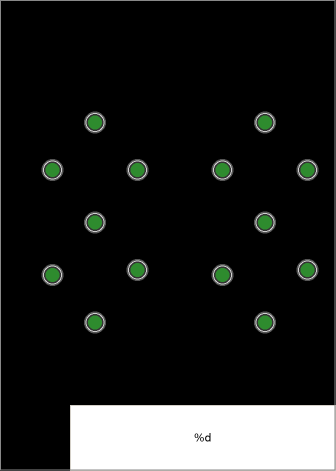
VISUALIZATION sevenSegmentDisplay  // 336x471
    Lamp1 (60,110 70x25), variable: sevenSegProg.digit1Decoder.decodedDigit[0], style: Lamp-Lamp1-Green
    Lamp1 (125,135 25x70), variable: sevenSegProg.digit1Decoder.decodedDigit[1], style: Lamp-Lamp1-Green
    Lamp1 (40,135 25x70), variable: sevenSegProg.digit1Decoder.decodedDigit[5], style: Lamp-Lamp1-Green
    Lamp1 (60,210 70x25), variable: sevenSegProg.digit1Decoder.decodedDigit[6], style: Lamp-Lamp1-Green
    Lamp1 (60,310 70x25), variable: sevenSegProg.digit1Decoder.decodedDigit[3], style: Lamp-Lamp1-Green
    Lamp1 (125,235 25x70), variable: sevenSegProg.digit1Decoder.decodedDigit[2], style: Lamp-Lamp1-Green
    Lamp1 (40,240 25x70), variable: sevenSegProg.digit1Decoder.decodedDigit[4], style: Lamp-Lamp1-Green
    Textfield (70,405 266x66), "%d", text variable: sevenSegProg.inputDigit
        OnMouseClick: write sevenSegProg.inputDigit via Default
    Lamp1 (230,110 70x25), variable: sevenSegProg.digit2Decoder.decodedDigit[0], style: Lamp-Lamp1-Green
    Lamp1 (295,135 25x70), variable: sevenSegProg.digit2Decoder.decodedDigit[1], style: Lamp-Lamp1-Green
    Lamp1 (210,135 25x70), variable: sevenSegProg.digit2Decoder.decodedDigit[5], style: Lamp-Lamp1-Green
    Lamp1 (230,210 70x25), variable: sevenSegProg.digit2Decoder.decodedDigit[6], style: Lamp-Lamp1-Green
    Lamp1 (230,310 70x25), variable: sevenSegProg.digit2Decoder.decodedDigit[3], style: Lamp-Lamp1-Green
    Lamp1 (295,235 25x70), variable: sevenSegProg.digit2Decoder.decodedDigit[2], style: Lamp-Lamp1-Green
    Lamp1 (210,240 25x70), variable: sevenSegProg.digit2Decoder.decodedDigit[4], style: Lamp-Lamp1-Green
END_VISUALIZATION

(* stored: Version 1.1.0.1, ProductVersion 3.1.4024.5
   Visu sevenSegmentDisplay: Id {7ccd3555-30e6-4730-b57c-7ce0a465806f} *)
